{attribute 'pack_mode':='1'}
TYPE ST_LightTower :
	STRUCT
		GREEN			: BOOL;
		RED				: BOOL;	
		YELLOW			: BOOL;	
		BLUE			: BOOL;
		WHITE			: BOOL;
		BEEPING			: BOOL;
	END_STRUCT
END_TYPE

(* stored: Version 1.1.0.1, ProductVersion 3.1.4024.12
   DUT ST_LightTower: Id {b7d456ca-295c-4f24-93f8-088f27a12216} *)
